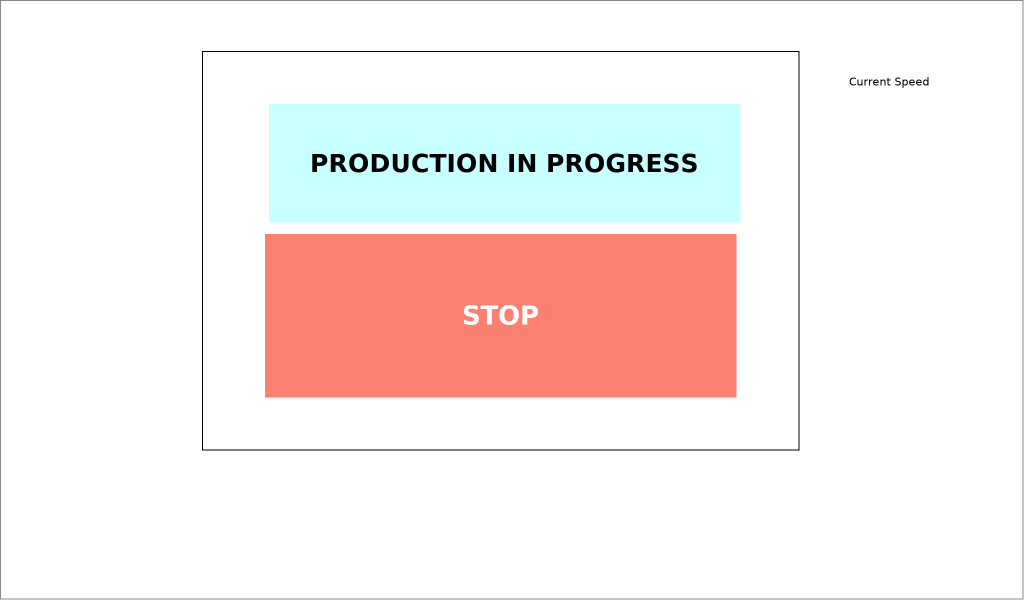
VISUALIZATION V_InfoMenu  // 1024x600
    RoundedRectangle (202,51 597x399)
    RoundedRectangle (268,103 473x120), "PRODUCTION IN PROGRESS"
    RoundedRectangle (264,233 473x165), "STOP"
        toggle GVL_Safety.eStopHMI
    Label (829,67 121x30), "Current Speed"
END_VISUALIZATION

(* stored: Version 1.1.0.1, ProductVersion 3.1.4024.15
   Visu V_InfoMenu: Id {a605f27f-6b24-0012-2ed8-5e678528cd71} *)
